PROGRAM P_Demo_F_BA_TimeStruct_TO_DateTime
VAR
    argTValue                      : TIMESTRUCT                    ; // tValue
    fnReturn                       : ST_BA_DateTime; // 返回值
END_VAR

// =============================================================================
// Tc3_BA2_Common.F_BA_TimeStruct_TO_DateTime 演示程序
// =============================================================================
// 场景：从 Windows 系统时间（`FB_LocalSystemTime` 返回 `TIMESTRUCT`）转成 BA 库的标准结构以便存入趋势数据库。
//
// 价值：一行 FC 替代手写逐字段 `dt.nYear := ts.wYear; dt.nMonth := ts.wMonth; ...` 等约 7 行映射。
//
// 验证：登录 PLC 后，按例程内变量在线写值；监视输出 / 返回值，结合 §1 功能
//       简述的预期行为对照（详见配套 .md 文档 §7 业务场景）。
//
// 验证步骤：
//   1. 右键 PLC 项目下 POUs 文件夹 → Add → Existing Item → 选本 .TcPOU 文件
//   2. 引用 Tc3_BA2_Common（References → Add library）
//   3. 编译 → 登录 → 运行；按上方『验证』指引在线写值观察
// =============================================================================

fnReturn := F_BA_TimeStruct_TO_DateTime(
    tValue                   := argTValue
);

END_PROGRAM

(* stored: Version 1.1.0.1, ProductVersion 3.1.4024.5
   POU P_Demo_F_BA_TimeStruct_TO_DateTime: Id {365a67b7-ff68-5871-9bf3-f400416286ed}, SpecialFunc None *)
